% RSLogix 500 project pump control with alarm and notifications.RSS, saved by version 8.30.00.16 %
PROJECT "AB"    % processor: Bul.1763 MicroLogix 1100 Series B %

PROGRAM FILES
  LAD 2 "MAIN"  4 rungs
  LAD 3 "ALARMS"  7 rungs
  LAD 4 "IO"  4 rungs
  LAD 5 "CONTROLS"  6 rungs

DATA FILES
  O0 OUTPUT  5 elements
  I1 INPUT  14 elements
  S2 STATUS  66 elements
  B3 BINARY  1 elements
  T4 TIMER  2 elements
  C5 COUNTER  1 elements
  R6 CONTROL  1 elements
  N7 INTEGER  1 elements
  F8 FLOAT  1 elements

LADDER 2 "MAIN"
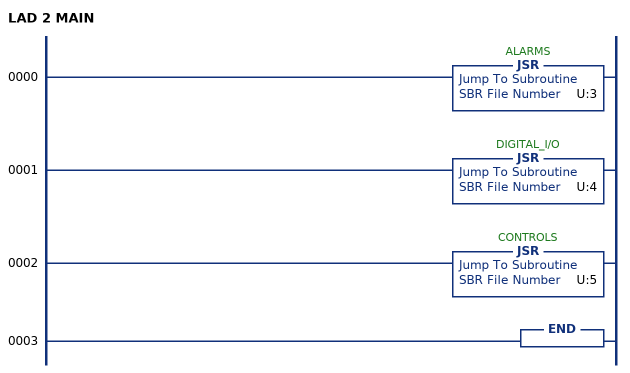
% Rung: 0 %  % edit flag set %
SOR JSR U:3 EOR
%   U:3  "ALARMS" %
% Rung: 1 %  % edit flag set %
SOR JSR U:4 EOR
%   U:4  "DIGITAL_I/O" %
% Rung: 2 %
SOR JSR U:5 EOR
%   U:5  "CONTROLS" %
% Rung: 3 %
SOR END EOR

LADDER 3 "ALARMS"
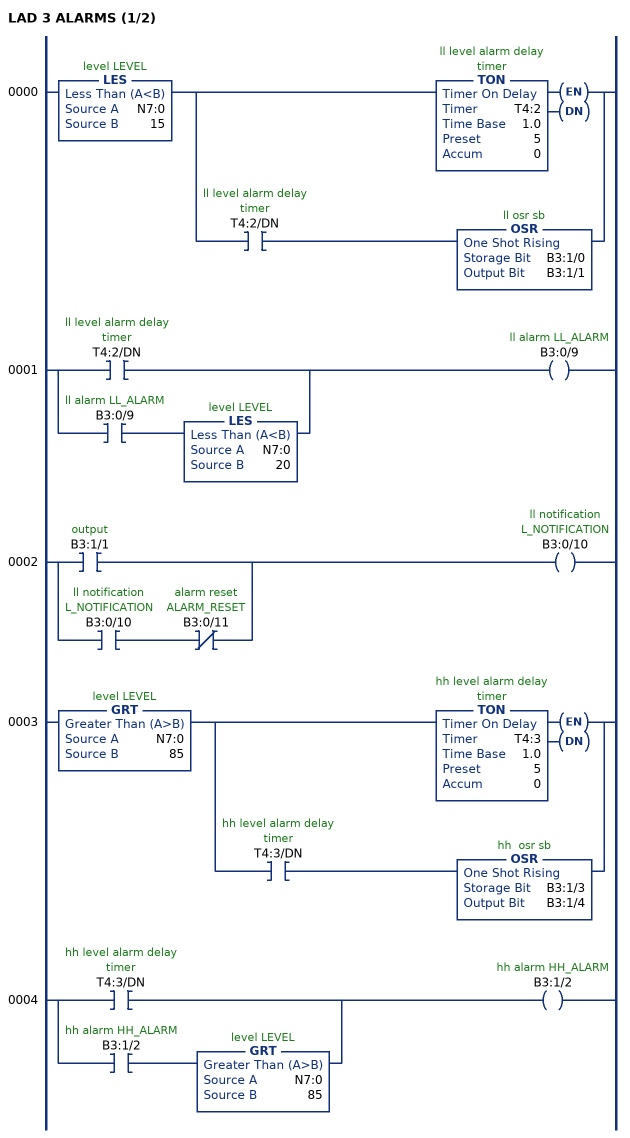
% Rung: 0 %  % edit flag set %
SOR LES N7:0 15 BST TON T4:2 1.0 5 0 NXB XIC T4:2/DN OSR B3:1/0 B3:1/1 BND EOR
%   N7:0  LEVEL  "level" %
%   T4:2  "ll level alarm delay timer" %
%   B3:1/0  "ll osr sb" %
%   B3:1/1  "output" %
% Rung: 1 %  % edit flag set %
SOR BST XIC T4:2/DN NXB XIC B3:0/9 LES N7:0 20 BND OTE B3:0/9 EOR
%   T4:2  "ll level alarm delay timer" %
%   B3:0/9  LL_ALARM  "ll alarm" %
%   N7:0  LEVEL  "level" %
% Rung: 2 %  % edit flag set %
SOR BST XIC B3:1/1 NXB XIC B3:0/10 XIO B3:0/11 BND OTE B3:0/10 EOR
%   B3:1/1  "output" %
%   B3:0/10  L_NOTIFICATION  "ll notification" %
%   B3:0/11  ALARM_RESET  "alarm reset" %
% Rung: 3 %  % edit flag set %
SOR GRT N7:0 85 BST TON T4:3 1.0 5 0 NXB XIC T4:3/DN OSR B3:1/3 B3:1/4 BND EOR
%   N7:0  LEVEL  "level" %
%   T4:3  "hh level alarm delay timer" %
%   B3:1/3  "hh  osr sb" %
%   B3:1/4  "output" %
% Rung: 4 %  % edit flag set %
SOR BST XIC T4:3/DN NXB XIC B3:1/2 GRT N7:0 85 BND OTE B3:1/2 EOR
%   T4:3  "hh level alarm delay timer" %
%   B3:1/2  HH_ALARM  "hh alarm" %
%   N7:0  LEVEL  "level" %

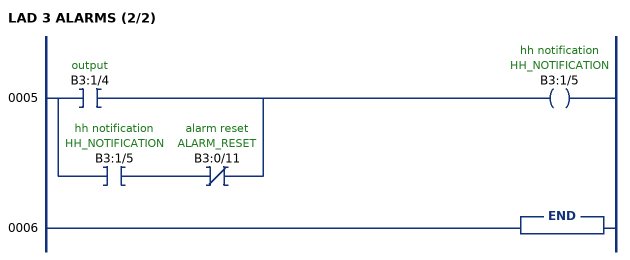
% Rung: 5 %  % edit flag set %
SOR BST XIC B3:1/4 NXB XIC B3:1/5 XIO B3:0/11 BND OTE B3:1/5 EOR
%   B3:1/4  "output" %
%   B3:1/5  HH_NOTIFICATION  "hh notification" %
%   B3:0/11  ALARM_RESET  "alarm reset" %
% Rung: 6 %
SOR END EOR

LADDER 4 "IO"
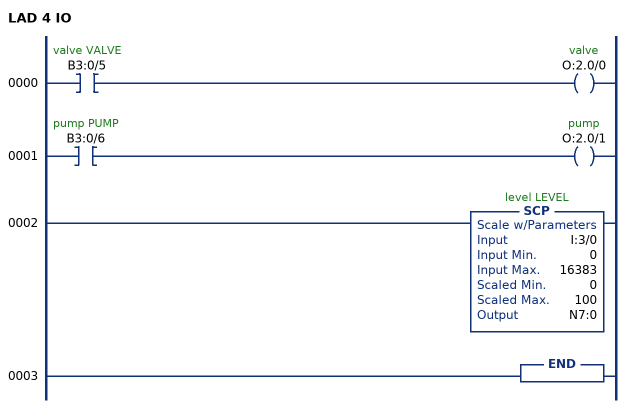
% Rung: 0 %
SOR XIC B3:0/5 OTE O:2.0/0 EOR
%   B3:0/5  VALVE  "valve" %
%   O:2.0/0  "valve" %
% Rung: 1 %
SOR XIC B3:0/6 OTE O:2.0/1 EOR
%   B3:0/6  PUMP  "pump" %
%   O:2.0/1  "pump" %
% Rung: 2 %  % edit flag set %
SOR SCP I:3/0 0 16383 0 100 N7:0 EOR
%   N7:0  LEVEL  "level" %
% Rung: 3 %
SOR END EOR

LADDER 5 "CONTROLS"
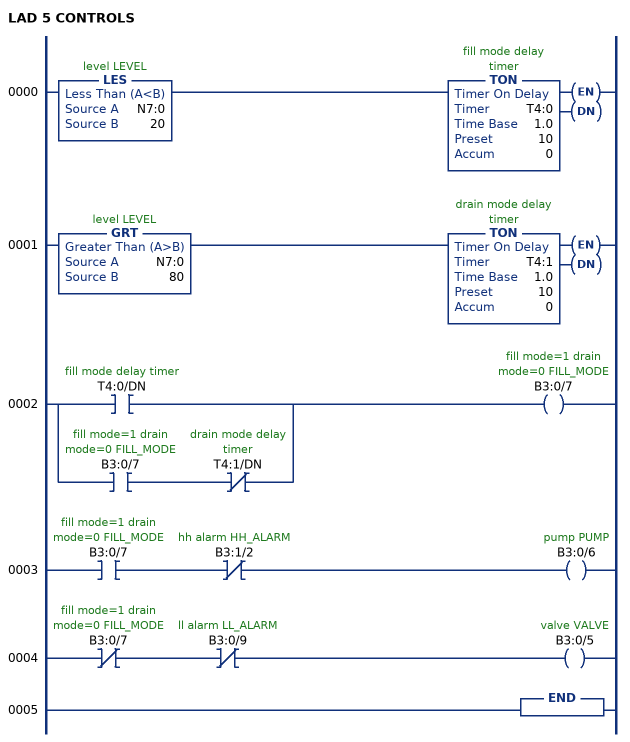
% Rung: 0 %  % edit flag set %
SOR LES N7:0 20 TON T4:0 1.0 10 0 EOR
%   N7:0  LEVEL  "level" %
%   T4:0  "fill mode delay timer" %
% Rung: 1 %  % edit flag set %
SOR GRT N7:0 80 TON T4:1 1.0 10 0 EOR
%   N7:0  LEVEL  "level" %
%   T4:1  "drain mode delay timer" %
% Rung: 2 %
SOR BST XIC T4:0/DN NXB XIC B3:0/7 XIO T4:1/DN BND OTE B3:0/7 EOR
%   T4:0/DN  "fill mode delay timer" %
%   B3:0/7  FILL_MODE  "fill mode=1 drain mode=0" %
%   T4:1/DN  "drain mode delay timer" %
% Rung: 3 %  % edit flag set %
SOR XIC B3:0/7 XIO B3:1/2 OTE B3:0/6 EOR
%   B3:0/7  FILL_MODE  "fill mode=1 drain mode=0" %
%   B3:1/2  HH_ALARM  "hh alarm" %
%   B3:0/6  PUMP  "pump" %
% Rung: 4 %  % edit flag set %
SOR XIO B3:0/7 XIO B3:0/9 OTE B3:0/5 EOR
%   B3:0/7  FILL_MODE  "fill mode=1 drain mode=0" %
%   B3:0/9  LL_ALARM  "ll alarm" %
%   B3:0/5  VALVE  "valve" %
% Rung: 5 %
SOR END EOR

OTHER DOCUMENTED ADDRESSES
  B3:0/0  LL_SWITCH  "L switch"
  B3:0/1  L_SWITCH  "L switch"
  B3:0/2  H_SWITCH  "H switch"
  B3:0/3  HH_SWITCH  "HH switch"
  B3:1/6  "alarm reset"
  I:1.0/0  "LL switch i/p"
  I:1.0/1  "L switch i/p"
  I:1.0/2  "H switch i/p"
  I:1.0/3  "HH_switch i/p"
  I:3.0/0  "level sensor input"

DATA TABLE (non-zero values as saved)
DATA T4
% .PRE .ACC %
% T4:0 % 10 0
% T4:1 % 10 0
